// TIA Portal V20 export
DATA_BLOCK "PNDevDiagInterface_X1"   // DB170
// stored: InstanceOfName LAF_typeDevDiagInterface, InstanceOfType UDT
"LAF_typeDevDiagInterface"
   // VAR
   //    globalInfoHmi : "LAF_typeDevDiagGlobal";
   //    devStateHmi { ExternalWritable := 'False'} : Array[0..256] of "LAF_typeDevDiagBasic";
   //    devStateUser { ExternalAccessible := 'False'; ExternalVisible := 'False'; ExternalWritable := 'False'} : Array[0..256] of "LAF_typeDevDiagState";
   // END_VAR
BEGIN
END_DATA_BLOCK
